TYPE
    OutputBase_10CEE7DE :
    STRUCT
    END_STRUCT
END_TYPE

(* stored: Version 1.1.0.1, ProductVersion 3.1.4024.12
   DUT OutputBase_10CEE7DE: Id {d4e7ad06-4b9a-0579-22dc-d6d53d00cfcf} *)
